FUNCTION_BLOCK FB_AutoGreaser EXTENDS FB_BaseDevice
VAR_INPUT
END_VAR
VAR_OUTPUT
END_VAR
VAR
END_VAR

END_FUNCTION_BLOCK

(* stored: Version 1.1.0.1, ProductVersion 3.1.4024.12
   POU FB_AutoGreaser: Id {51e4fc2c-b6de-4b44-a745-7ffb6a961ee5}, SpecialFunc None *)
